(* PLC project Generated.project, CODESYS CODESYS V3.5 SP19 Patch 1 *)
(* stored: creationDateTime 2026-11-18T01:43:05.022303, modificationDateTime 2026-11-18T01:43:05.022303 *)

(* values of E_MachineHomingTxState: HX0_REPOS: Repos : N1 libre bloque si NOT Homed, M3 bloque N1/SEMI, attente 5s BP joy N1 ou BtnStart N2; HX1_BUCKET_PREPARE: M2 seul palier 1, ouv + ferm sans butees soft, garde continue 20s + decompte, BtnValidate neutre; HX2_CLIMB_TO_TOP: Couple M1+M2 palier 1 : montee lente + detente 2s max/geste, viser avant TOP sans toucher; HX3_TOP_CLEARANCE: Contact TOP = perdu/surcourse -> montee interdite, descente ~4s apres relachement TOP -> retour HX1; HX4_FINAL_CONFIRM: Arret avant TOP + avertissement -> BtnValidate neutre -> preset 8.5m M1+M2 + CommitClose -> Homed; HX7_FAILED: Echec / abandon : coupure mouvements, purge etats, attente Reset conscient *)

{attribute 'qualified_only'}
{attribute 'strict'}
TYPE E_MachineHomingTxState : (HX0_REPOS := 0, HX1_BUCKET_PREPARE := 1, HX2_CLIMB_TO_TOP := 2, HX3_TOP_CLEARANCE := 3, HX4_FINAL_CONFIRM := 4, HX7_FAILED := 5);
END_TYPE
